// TwinCAT 3 PLC project lclc_plc_neh_n2
// ProgramVersion: 3.1.4022.7
// libraries:
//   LCLS General, * (SLAC)
//   Tc2_Standard, * (Beckhoff Automation GmbH)
//   Tc2_System, * (Beckhoff Automation GmbH)
//   Tc3_Module, * (Beckhoff Automation GmbH)
// project tree:
//   DUTs/ ENUM_LED_MODES.TcDUT (not stored)
//   / PlcTask.TcTTO (not stored)
//   POUs/ FB_VALVE_RELAY.TcPOU, MAIN.TcPOU

// ---- POUs/FB_VALVE_RELAY.TcPOU
FUNCTION_BLOCK FB_VALVE_RELAY 
VAR_IN_OUT
END_VAR
VAR_INPUT
END_VAR
VAR_OUTPUT
	bTimerQ : BOOL;
END_VAR
VAR
	b_open : BOOL; // control variable
	// EL2624 Relayu Logic Here

	rawOutputRelayChan1 AT %Q*: BOOL;
	rawOutputRelayChan3 AT %Q*: BOOL;
	bCloseRBV AT %I* : BOOL;
	bOpenRBV AT %I* : BOOL;
	bMovingRBV AT %I* : BOOL;
	
	tActuateTime : TIME := T#24h;
	iState: INT;
	fbValveTimer : TON;
END_VAR


fbValveTimer(IN:=TRUE, PT:=tActuateTime);

CASE iState OF
    0: // INIT
    fbValveTimer(IN:=FALSE); //RESTART TIMER
    iState := 1;

    1: // NOMINAL
	ACTUATE_VALVE(b_open); 
 
	IF fbValveTimer.Q THEN iState := 2; END_IF
	
	2: // Do the opposite of current valve state
	IF bCloseRBV THEN ACTUATE_VALVE(TRUE);END_IF
	IF bOpenRBV THEN ACTUATE_VALVE(FALSE);END_IF
	IF bMovingRBV THEN iState := 3; END_IF; // Only transition when we have started to move
	
	3: // Go back to init to reset timer and return valve to previous state.
	IF NOT bMovingRBV THEN iState := 0; END_IF;

END_CASE

bTimerQ := fbValveTimer.Q;

METHOD ACTUATE_VALVE : BOOL
VAR_INPUT
	b_open: BOOL;
END_VAR
IF b_open THEN
	rawOutputRelayChan1 := FALSE;
	rawOutputRelayChan3 := TRUE;
ELSE
	rawOutputRelayChan1 := TRUE;
	rawOutputRelayChan3 := FALSE;
END_IF
END_METHOD

END_FUNCTION_BLOCK

// ---- POUs/MAIN.TcPOU
PROGRAM MAIN
VAR
    fbGetmA: FB_AnalogInput;
    fmA: LREAL;
    {attribute 'TcLinkTo' := 'TIID^Device 1 (EtherCAT)^Term 1 (EK1200)^Term 2 (EL3052)^AI Standard Channel 1^Value'}
    rawInputmA AT %I*: INT;

	fPress : LREAL;
	
	bInduceButton AT %I*	: BOOL;
	bFinishExchangeButton AT %I*	: BOOL;
	fMinPressureThresh 		: LREAL;
	fMinMassThresh			: LREAL;
	fWarningThresh: LREAL;
	eLEDMode : ENUM_LED_MODES;
	bValveTimerQ : BOOL;


    {attribute 'pytmc' := 'pv: XBD:N2:MAX_MASS'}
    maxMass: LREAL;
    {attribute 'pytmc' := 'pv: XBD:N2:MIN_MASS'}
    minMass: LREAL;
    {attribute 'pytmc' := 'pv: XBD:N2:CURRENT_MASS'}
    fMassofGas: LREAL;

    {attribute 'pytmc' := 'pv: XBD:N2:LOW_LEVEL'}
    fMassLowLevl : LREAL := maxMass / 2;
    bMassIsLow : BOOL := FALSE;

	{attribute 'TcLinkTo' := '
		.rawOutputRelayChan1 := TIID^Device 1 (EtherCAT)^Term 1 (EK1200)^Term 5 (EL2624)^Channel 1^Output;
		.rawOutputRelayChan3 := TIID^Device 1 (EtherCAT)^Term 1 (EK1200)^Term 5 (EL2624)^Channel 2^Output;
		.bCloseRBV := TIID^Device 1 (EtherCAT)^Term 1 (EK1200)^Term 6 (EL1004)^Channel 1^Input;
		.bOpenRBV := TIID^Device 1 (EtherCAT)^Term 1 (EK1200)^Term 6 (EL1004)^Channel 2^Input;
		.bMovingRBV := TIID^Device 1 (EtherCAT)^Term 1 (EK1200)^Term 6 (EL1004)^Channel 3^Input;
	'}
    fbValveRelay : FB_VALVE_RELAY;

    bInit : BOOL := TRUE;
    iState : INT  := 0;

END_VAR

IF bInit THEN
    maxMass := 500;
    minMass := 0;
    bInit := FALSE;
END_IF

fbValveRelay(bTimerQ=>bValveTimerQ);
//fbLightTower(iLIGHT_MODE);

fbGetmA(
    iRaw := rawInputmA,
    iTermBits := 12,
    fTermMax := 20,
    fTermMin := 4,
    fReal => fmA
);

fMassofGas := (fmA - 4.0) / 16.0 * maxMass + minMass;

CASE iState OF
	-1: // INIT
	fbValveRelay.ACTUATE_VALVE(FALSE);
	 IF ((fPress > fMinPressureThresh) AND (fmA > fMinMassThresh)) THEN fbValveRelay.ACTUATE_VALVE(TRUE); END_IF
	iState := 0;
	
    0: // Nominal
    IF  ((fPress < fMinPressureThresh) OR (fmA < fMinMassThresh) OR (bInduceButton)) THEN
		// TURN LIGHT RED
        iState := 1;
		fbValveRelay.ACTUATE_VALVE(FALSE);
    END_IF
	
	IF (fmA < fWarningThresh) THEN 
		// TURN ON YELLOW LIGHT
	END_IF
	
	IF(bValveTimerQ) THEN
		// FLASH YELLO LIGHT
	END_IF
	
    1: // EXCHANGE MODE
	IF (bInduceButton) THEN
		// TURN FLASHY RED
	END_IF
	IF  ((bFinishExchangeButton)) THEN
        iState := -1;
		// TURN OFF RED LIGHT
    END_IF
	
	

END_CASE

END_PROGRAM
